{attribute 'GeneratedUsingTerminal: EPP7342-0002-0016'}
{attribute addProperty BoxType "EPP7342-0002-0016"}
{attribute addProperty Id "Enable_latch_extern_on_positive_edgeBOOL1Set_counterBOOL1Enable_latch_extern_on_negative_edgeBOOL1"}
{attribute addProperty CRC "4052334391"}
{attribute addProperty Size "3"}
TYPE Control_F189B737 :
STRUCT
	{attribute addProperty Name "Enable_latch_extern_on_positive_edge"}
	Enable_latch_extern_on_positive_edge : BOOL;
	{attribute addProperty Name "Set_counter"}
	Set_counter : BOOL;
	{attribute addProperty Name "Enable_latch_extern_on_negative_edge"}
	Enable_latch_extern_on_negative_edge : BOOL;
END_STRUCT
END_TYPE

(* stored: Version 1.2.0.0, ProductVersion 3.1.4024.9
   DUT Control_F189B737: Id {f1acd25f-7234-4c5a-8758-58cf9ed2d2da} *)
